FUNCTION F_InRange : BOOL
VAR_INPUT
	fValue			: LREAL;	//11.5
	fLowerLimit		: LREAL;	//10
	fUpperLimit		: LREAL;	//12	
END_VAR
VAR
	fTempUl			: LREAL;
	fTempLl			: LREAL;
END_VAR

F_InRange:=(fValue >= fLowerLimit) AND (fValue <= fUpperLimit);

END_FUNCTION

(* stored: Version 1.1.0.1, ProductVersion 3.1.4024.11
   POU F_InRange: Id {87b424eb-3d5d-4f4a-9f7c-4ea9b0b575fd}, SpecialFunc None *)
